(* CODESYS project DemoLibrary.library
   Title: DemoBasicLibrary
   Version: 1.0.0
   Placeholder: DemoBasicLibrary
   Company: GithubExamples

Project tree, tasks and I/O mapping:
  function block MyFunctionBlock [ST]
*)

// MyFunctionBlock
FUNCTION_BLOCK MyFunctionBlock
VAR
END_VAR

END_FUNCTION_BLOCK
